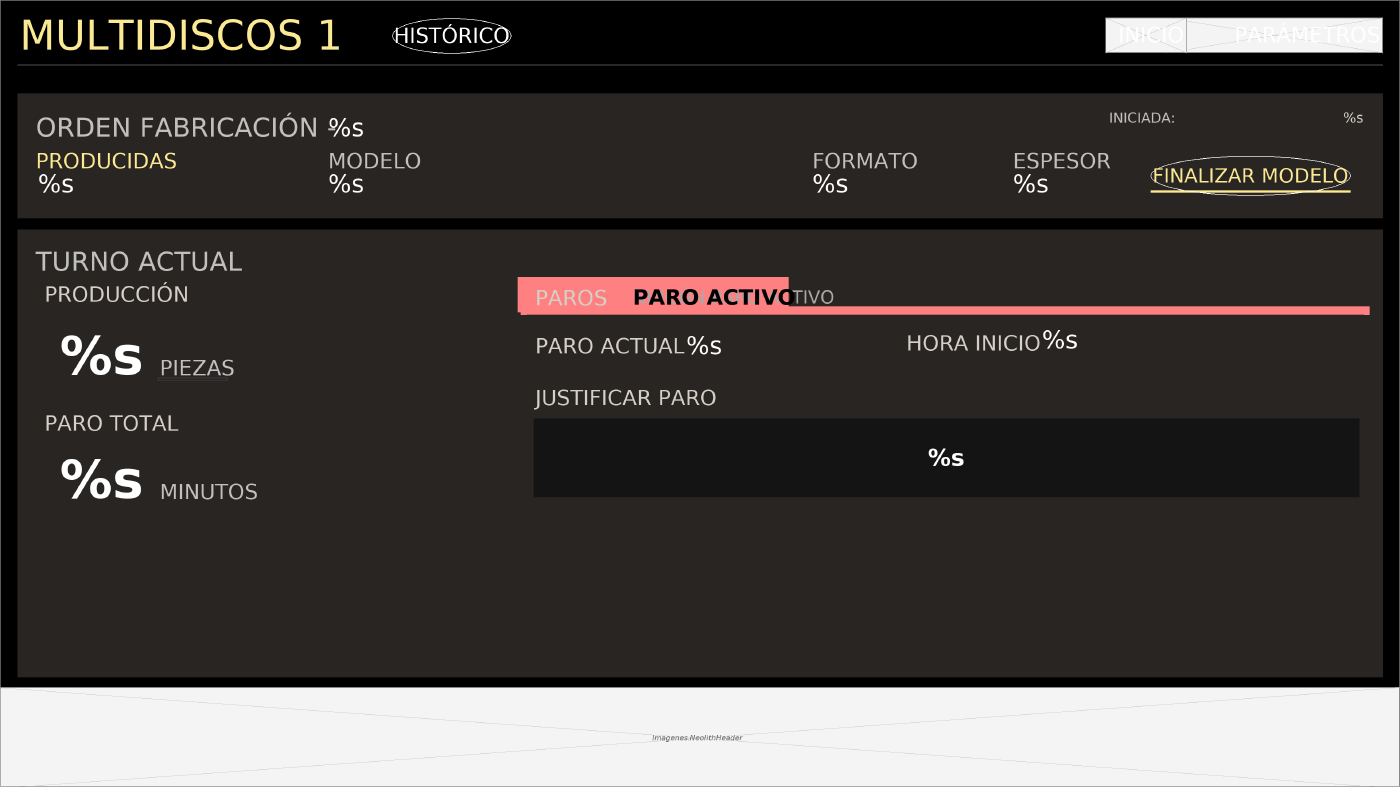
VISUALIZATION Home_Multidis1  // 1920x1080
    Ellipse (1559,1109 456x77), "Fin de producción del modelo"
        OnMouseClick: OpenDialog Dialog=V_Emerg_Fin_Prod_Md1, OpenModal=True, OpenCentered=True
    Rectangle (2270,679 183x30), "%s", text variable: FuncParoNodoMultidiscos.Funci_Multidiscos1.H_InParo_Ftc, invisible if: FuncParoNodoMultidiscos.Funci_Multidiscos1.M_SinParo_Ftc
    Label (2034,678 239x30), "Hora Inicio del paro", invisible if: FuncParoNodoMultidiscos.Funci_Multidiscos1.M_SinParo_Ftc
    Rectangle (2270,737 192x30), "%s", text variable: FuncParoNodoMultidiscos.Funci_Multidiscos1.Min_Parado_Ftc, invisible if: FuncParoNodoMultidiscos.Funci_Multidiscos1.M_SinParo_Ftc
    Label (2069,737 204x30), "Minutos Parado", invisible if: FuncParoNodoMultidiscos.Funci_Multidiscos1.M_SinParo_Ftc
    Label (2029,792 244x30), "Tiempo entre Piezas"
    Label (2018,828 255x62), "Tiempo entre Piezas Anterior"
    Rectangle (2532,486 183x123), "%s", text variable: FuncParoNodoMultidiscos.Funci_Multidiscos1.Cont_Piezas_Ftc
    Rectangle (2270,792 192x30), "%s", text variable: FuncParoNodoMultidiscos.Funci_Multidiscos1.t_Entre_Piez_Ftc
    Rectangle (2270,844 192x30), "%s", text variable: FuncParoNodoMultidiscos.Funci_Multidiscos1.t_Entr_Piez_Ante_Ftc
    Label (2029,582 326x30), "En producción todo OK", invisible if: FuncParoNodoMultidiscos.Funci_Multidiscos1.MParo_Ftc
    Label (2047,507 235x59), "Línea en paro", invisible if: FuncParoNodoMultidiscos.Funci_Multidiscos1.M_SinParo_Ftc
    Label (2424,368 354x119), "Número de losas"
    Rectangle (234,1309 1380x154), "%s", text variable: FuncParoNodoMultidiscos.Funci_Multidiscos1.S_Justi_Paro_Ftc, invisible if: FuncParoNodoMultidiscos.Funci_Multidiscos1.M_SinParo_Ftc
        OnMouseDown: write the text variable via Edit
    Label (25,1090 1381x106), "JUSTIFICAR EL PARO ACTUAL", invisible if: FuncParoNodoMultidiscos.Funci_Multidiscos1.M_SinParo_Ftc
    Image (893,-598 250x250), invisible if: FuncParoNodoMultidiscos.Funci_Multidiscos1.M_SinParo_Ftc, image: ImagePool.Exclamación
    Rectangle (24,88 1872x2)
    Label (24,16 514x64), "MULTIDISCOS 1"
    Image (1600,24 296x48), "PARÁMETROS"
        OnMouseClick: change screen: Ajustes_CorteH4
    Image (1516,24 111x48), "INICIO"
        OnMouseClick: change screen: Home_Sel_Maq
    Ellipse (538,25 163x48), "HISTÓRICO"
        OnMouseClick: change screen: HistTablaTablas_Ch4
    Rectangle (24,128 1872x171)
    Label (46,148 390x54), "ORDEN FABRICACIÓN -"
    Rectangle (1573,147 300x30), "%s", text variable: FuncParoNodoMultidiscos.sFechaInicModeloTab_MD1
    Label (1518,147 99x30), "INICIADA:"
    Rectangle (447,232 671x40), "%s", text variable: FuncParoNodoMultidiscos.sModeloActualTabla_MD1
    Rectangle (1386,232 120x40), "%s", text variable: FuncParoNodoMultidiscos.sEspesorActualTabla_MD1
    Rectangle (1111,232 321x40), "%s", text variable: FuncParoNodoMultidiscos.sFormatoActualTabla_MD1
    Label (447,203 487x36), "MODELO"
    Label (1111,203 156x36), "FORMATO"
    Label (1386,203 156x36), "ESPESOR"
    Rectangle (447,155 321x40), "%s", text variable: FuncParoNodoCorteH4Remote1.sFormatoActualTabla
    Label (46,203 199x36), "PRODUCIDAS"
    Rectangle (49,232 248x40), "%s", text variable: FuncParoNodoCorteH4Remote1.sEspesorActualTabla
    Group (1578,214 274x54)
        Rectangle (0,47 274x3)
        Ellipse (0,0 274x54), "FINALIZAR MODELO"
            OnMouseClick: OpenDialog Dialog=V_Emerg_Fin_Prod_Md1, OpenModal=True, OpenCentered=True
    Rectangle (24,315 1872x614)
    Rectangle (1426,451 401x30), "%s", text variable: FuncParoNodoMultidiscos.Funci_Multidiscos1.H_InParo_Ftc, invisible if: FuncParoNodoMultidiscos.Funci_Multidiscos1.M_SinParo_Ftc
    Rectangle (938,459 192x30), "%s", text variable: FuncParoNodoMultidiscos.Funci_Multidiscos1.Min_Parado_Ftc, invisible if: FuncParoNodoMultidiscos.Funci_Multidiscos1.M_SinParo_Ftc
    Rectangle (732,574 1132x108), "%s", text variable: FuncParoNodoMultidiscos.Funci_Multidiscos1.S_Justi_Paro_Ftc, invisible if: FuncParoNodoMultidiscos.Funci_Multidiscos1.M_SinParo_Ftc
        OnMouseDown: write the text variable via Edit
    Label (46,332 390x54), "TURNO ACTUAL"
    Label (58,386 199x36), "PRODUCCIÓN"
    Label (731,457 261x36), "PARO ACTUAL", invisible if: FuncParoNodoMultidiscos.Funci_Multidiscos1.M_SinParo_Ftc
    Label (1240,453 261x36), "HORA INICIO", invisible if: FuncParoNodoMultidiscos.Funci_Multidiscos1.M_SinParo_Ftc
    Rectangle (79,444 183x88), "%s", text variable: FuncParoNodoMultidiscos.Funci_Multidiscos1.Cont_Piezas_Ftc
    Label (216,487 106x36), "PIEZAS"
    Rectangle (216,518 96x4), colour toggle: FuncParoNodoMultidiscos.Funci_Multidiscos1.Fotocelula
    Label (731,528 261x36), "JUSTIFICAR PARO", invisible if: FuncParoNodoMultidiscos.Funci_Multidiscos1.M_SinParo_Ftc
    Group (710,380 1168x48), invisible if: FuncParoNodoMultidiscos.Funci_Multidiscos1.M_SinParo_Ftc
        Rectangle (4,44 1164x4)
        Rectangle (0,0 371x48)
        Label (21,11 199x36), "PAROS"
        Label (155,13 326x30), "NINGÚN PARO ACTIVO", invisible if: FuncParoNodoCorteH4Remote1.Funci_CortHum4.MParo_Ftc
        Label (155,13 235x30), "PARO ACTIVO", invisible if: FuncParoNodoCorteH4Remote1.Funci_CortHum4.M_SinParo_Ftc
    Label (58,563 261x36), "PARO TOTAL"
    Rectangle (79,614 183x88), "%s", text variable: FuncParoNodoCorteH4Remote1.Funci_CortHum4.Cont_Piezas_Ftc
    Label (216,657 142x36), "MINUTOS"
    Image (-7,943 1927x139), image: Imagenes.NeolithHeader
END_VISUALIZATION

(* stored: Version 1.1.0.1, ProductVersion 3.1.4024.12
   Visu Home_Multidis1: Id {5948937d-8aea-4ee4-b087-572bc7a5e62b} *)
